(* PLC project CoDeSys External Library Template, WAGO e!COCKPIT e!COCKPIT, author 3S - Smart Software Solutions GmbH *)
(* stored: creationDateTime 2019-10-29T12:22:40.4593344, version 3.5.5.30, modificationDateTime 2019-10-24T14:40:07.960949, organization 3S - Smart Software Solutions GmbH *)
(* Library project template with all possible element types, docu and a sample project structure *)

(* values of enumPPPSSilownikSABpServiceFlag: BrakDzialan: Brak rozkazu; TrybLetni: Rozkaz ustwienia trybu letniego; ZamkniecieZaworu: Rozkaz zamknięcia zaworu; OtwarcieZaworu: Rozkaz otwarcia zaworu; PozycjaGorna: Rozkaz pozycji górnej trzpienia (pozycja do transportu) - po jego uruchomieniu wymagana ponowna kalibracja; KalibracjaSilownika: Rozkaz uruchomienia sekwencji inicjalizacji siłownika *)

(* Autor: Paweł Kąkol, 2018-09-04-PK Prawa majątkowe: Solwena Sp. z o.o., Aktualizacje: Opis: enum służy do obsługi flagi serwisowej siłownika SAB+ (HRU0) na budynkach PPP Sopot (ENGIE) *)
{attribute 'qualified_only'}
{attribute 'strict'}
TYPE enumPPPSSilownikSABpServiceFlag : (BrakDzialan := 0, TrybLetni := 1, ZamkniecieZaworu := 2, OtwarcieZaworu := 3, PozycjaGorna := 4, KalibracjaSilownika := 5);
END_TYPE
